FUNCTION_BLOCK MissingKeyDeserializationError_TestSuite EXTENDS TcUnit.FB_TestSuite

TestAccept();
TestErrorType();
TestIsSameAsWithSameErrors();
TestIsSameAsWithDifferentErrors();
TestMessage();
TestSerializeWith();

METHOD PUBLIC TestAccept
VAR
	error : MissingKeyDeserializationError('testKey');
	visitor : MockErrorVisitor(ExpectedError := error);
END_VAR
TEST('TestAccept');

error.Accept(visitor);

AssertTrue(
	Condition := visitor.VisitedCorrectError,
	Message := 'Did not invoke VisitError on the visitor'
);

TEST_FINISHED();
END_METHOD

METHOD PUBLIC TestErrorType
VAR
	error : MissingKeyDeserializationError('testKey');
END_VAR
TEST('TestErrorType');

AssertEquals_String(
	Actual := error.ErrorType,
	Expected := 'MISSING_KEY_DESERIALIZATION_ERROR',
	Message := 'Did not return the expected ErrorType'
);

TEST_FINISHED();
END_METHOD

METHOD PUBLIC TestIsSameAsWithDifferentErrors
VAR
	error1 : MissingKeyDeserializationError('testKey');
	error2 : MockError(MockErrorType:='ERROR_TYPE_B',MockMessage:='Message 2');
END_VAR
TEST('TestIsSameAsWithDifferentErrors');

AssertFalse(
	Condition := error1.IsSameAs(error2),
	Message := 'Did not correctly identify errors as being different type'
);

TEST_FINISHED();
END_METHOD

METHOD PUBLIC TestIsSameAsWithSameErrors
VAR
	error1 : MissingKeyDeserializationError('testKey');
	error2 : MockError(MockErrorType:='MISSING_KEY_DESERIALIZATION_ERROR',MockMessage:='Message');
END_VAR
TEST('TestIsSameAsWithSameErrors');

AssertTrue(
	Condition := error1.IsSameAs(error2),
	Message := 'Did not correctly identify errors as being the same type'
);

TEST_FINISHED();
END_METHOD

METHOD PUBLIC TestMessage
VAR
	error : MissingKeyDeserializationError('testKey');
END_VAR
TEST('TestMessage');

AssertEquals_String(
	Actual := error.Message,
	Expected := 'Deserialization Failed, Missing Key : testKey',
	Message := 'Did not return the expected Message'
);

TEST_FINISHED();
END_METHOD

METHOD PUBLIC TestSerializeWith
VAR
	error : MissingKeyDeserializationError('testKey');
	serializer : MockJsonSerializer;
	result : T_MAXSTRING;
END_VAR
TEST('TestSerializeWith');

error.SerializeWith(serializer);
serializer.TryGetSerializedData(ADR(result), SIZEOF(result));

AssertEquals_String(
	Actual := result,
	Expected := '{"errorType":"MISSING_KEY_DESERIALIZATION_ERROR","message":"Deserialization Failed, Missing Key : testKey"}',
	Message := 'Did not serialize correctly'
);

TEST_FINISHED();
END_METHOD

END_FUNCTION_BLOCK

(* stored: Version 1.1.0.1, ProductVersion 3.1.4024.12
   POU MissingKeyDeserializationError_TestSuite: Id {f652332c-2aec-0ff1-3e0a-0597b8cba29b}, SpecialFunc None
   Method TestAccept: Id {e633dd56-4d0b-0092-280a-9aca1128ce80}
   Method TestErrorType: Id {82bb96a7-6380-0a94-109b-4df216c9d813}
   Method TestIsSameAsWithDifferentErrors: Id {9c6bac54-9a4b-001a-1859-2430cdb0d48b}
   Method TestIsSameAsWithSameErrors: Id {ae0f6b18-67c3-0ffb-0445-d4010142aaba}
   Method TestMessage: Id {df5ce696-925e-0f26-2c56-0b0fe135e42e}
   Method TestSerializeWith: Id {c54f94be-572a-0c26-144c-0ec64c5a591e} *)
